FUNCTION_BLOCK goToRelPos (* Composite Function Block Type *)
  (* Standard: 61499-2 *)
  (* Version 1.0, 2019-05-27, Promok *)
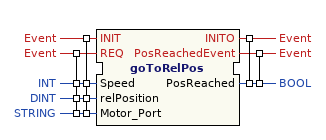
  EVENT_INPUT
    INIT WITH Speed, Motor_Port, relPosition; (* Initialization Request *)
    REQ WITH Speed, Motor_Port, relPosition; (* Normal Execution Request *)
  END_EVENT
  EVENT_OUTPUT
    INITO WITH PosReached; (* Initialization Confirm *)
    PosReachedEvent WITH PosReached;
  END_EVENT
  VAR_INPUT
    Speed : INT;
    relPosition : DINT;
    Motor_Port : STRING;
  END_VAR
  VAR_OUTPUT
    PosReached : BOOL;
  END_VAR
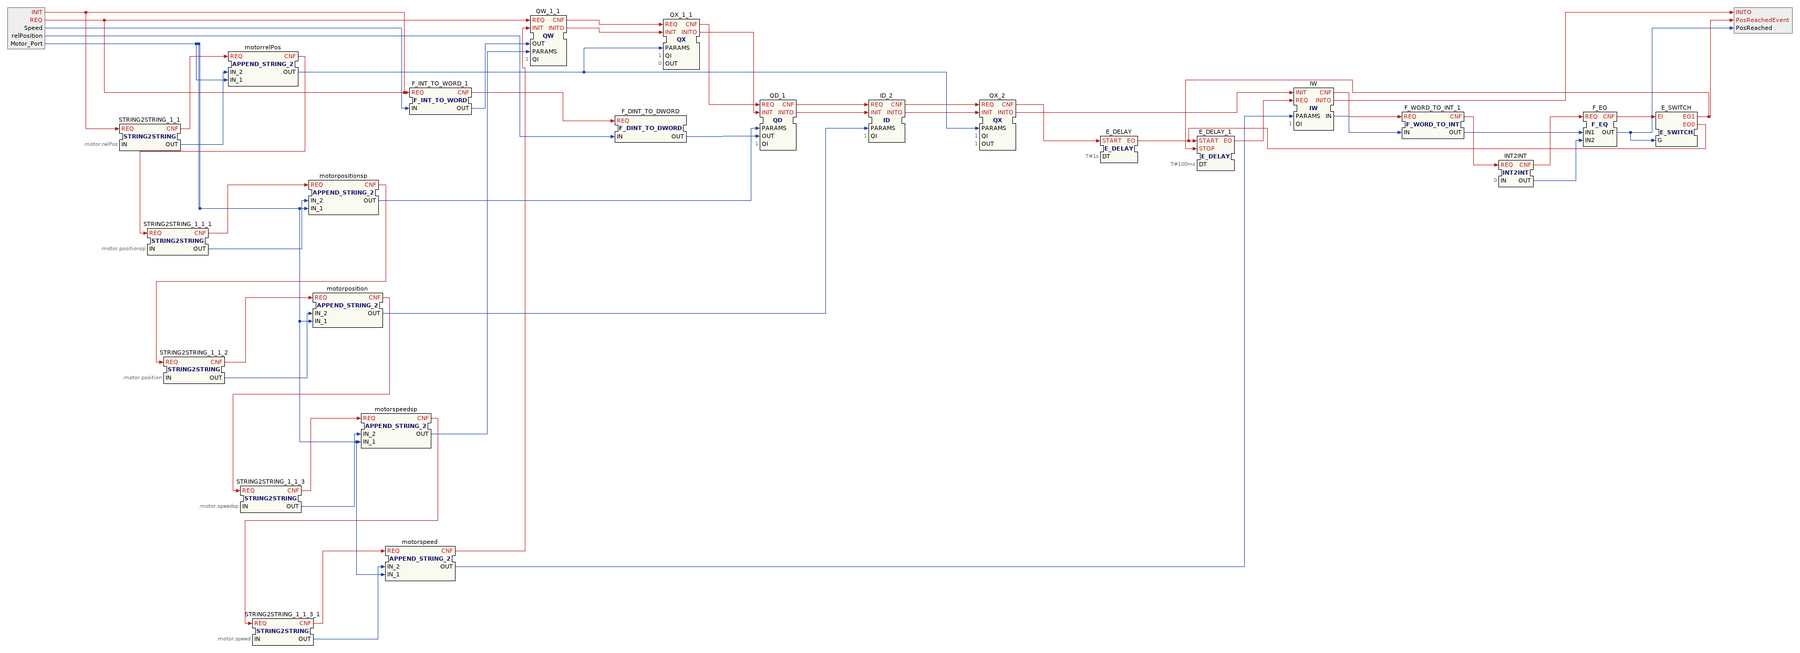
  FBS
    QX_1_1 : QX(QI := 1, OUT := 0);
    QW_1_1 : QW(QI := 1);
    QD_1 : QD(QI := 1);
    F_INT_TO_WORD_1 : F_INT_TO_WORD;
    ID_2 : ID(QI := 1);
    QX_2 : QX(QI := 1, OUT := 1);
    STRING2STRING_1_1 : STRING2STRING(IN := .motor.relPos);
    motorrelPos : APPEND_STRING_2;
    STRING2STRING_1_1_1 : STRING2STRING(IN := .motor.positionsp);
    motorpositionsp : APPEND_STRING_2;
    STRING2STRING_1_1_2 : STRING2STRING(IN := .motor.position);
    motorposition : APPEND_STRING_2;
    STRING2STRING_1_1_3 : STRING2STRING(IN := .motor.speedsp);
    motorspeedsp : APPEND_STRING_2;
    F_DINT_TO_DWORD : F_DINT_TO_DWORD;
    STRING2STRING_1_1_3_1 : STRING2STRING(IN := .motor.speed);
    motorspeed : APPEND_STRING_2;
    IW : IW(QI := 1);
    F_WORD_TO_INT_1 : F_WORD_TO_INT;
    E_DELAY : E_DELAY(DT := T#1s);
    F_EQ : F_EQ;
    INT2INT : INT2INT(IN := 0);
    E_SWITCH : E_SWITCH;
    E_DELAY_1 : E_DELAY(DT := T#100ms);
  END_FBS
  EVENT_CONNECTIONS
    QW_1_1.CNF TO QX_1_1.REQ;
    QW_1_1.INITO TO QX_1_1.INIT;
    QD_1.CNF TO ID_2.REQ;
    QX_1_1.CNF TO QD_1.REQ;
    QX_1_1.INITO TO QD_1.INIT;
    QD_1.INITO TO ID_2.INIT;
    STRING2STRING_1_1.CNF TO motorrelPos.REQ;
    STRING2STRING_1_1_1.CNF TO motorpositionsp.REQ;
    STRING2STRING_1_1_2.CNF TO motorposition.REQ;
    INIT TO STRING2STRING_1_1.REQ;
    motorrelPos.CNF TO STRING2STRING_1_1_1.REQ;
    motorpositionsp.CNF TO STRING2STRING_1_1_2.REQ;
    STRING2STRING_1_1_3.CNF TO motorspeedsp.REQ;
    motorposition.CNF TO STRING2STRING_1_1_3.REQ;
    REQ TO F_INT_TO_WORD_1.REQ;
    REQ TO QW_1_1.REQ;
    INIT TO F_INT_TO_WORD_1.REQ;
    F_INT_TO_WORD_1.CNF TO F_DINT_TO_DWORD.REQ;
    motorspeed.CNF TO QW_1_1.INIT;
    motorspeedsp.CNF TO STRING2STRING_1_1_3_1.REQ;
    STRING2STRING_1_1_3_1.CNF TO motorspeed.REQ;
    IW.CNF TO F_WORD_TO_INT_1.REQ;
    F_WORD_TO_INT_1.CNF TO INT2INT.REQ;
    INT2INT.CNF TO F_EQ.REQ;
    QX_2.CNF TO E_DELAY.START;
    ID_2.CNF TO QX_2.REQ;
    ID_2.INITO TO QX_2.INIT;
    IW.INITO TO INITO;
    QX_2.INITO TO IW.INIT;
    F_EQ.CNF TO E_SWITCH.EI;
    E_SWITCH.EO1 TO PosReachedEvent;
    E_DELAY.EO TO E_DELAY_1.START;
    E_DELAY_1.EO TO IW.REQ;
    E_SWITCH.EO1 TO E_DELAY_1.STOP;
    E_SWITCH.EO0 TO E_DELAY_1.START;
  END_CONNECTIONS
  DATA_CONNECTIONS
    F_INT_TO_WORD_1.OUT TO QW_1_1.OUT;
    STRING2STRING_1_1.OUT TO motorrelPos.IN_2;
    STRING2STRING_1_1_1.OUT TO motorpositionsp.IN_2;
    STRING2STRING_1_1_2.OUT TO motorposition.IN_2;
    Motor_Port TO motorrelPos.IN_1;
    Motor_Port TO motorpositionsp.IN_1;
    Motor_Port TO motorposition.IN_1;
    STRING2STRING_1_1_3.OUT TO motorspeedsp.IN_2;
    Motor_Port TO motorspeedsp.IN_1;
    motorspeedsp.OUT TO QW_1_1.PARAMS;
    motorrelPos.OUT TO QX_1_1.PARAMS;
    motorpositionsp.OUT TO QD_1.PARAMS;
    motorrelPos.OUT TO QX_2.PARAMS;
    motorposition.OUT TO ID_2.PARAMS;
    F_DINT_TO_DWORD.OUT TO QD_1.OUT;
    relPosition TO F_DINT_TO_DWORD.IN;
    Speed TO F_INT_TO_WORD_1.IN;
    STRING2STRING_1_1_3_1.OUT TO motorspeed.IN_2;
    Motor_Port TO motorspeed.IN_1;
    IW.IN TO F_WORD_TO_INT_1.IN;
    F_WORD_TO_INT_1.OUT TO F_EQ.IN1;
    motorspeed.OUT TO IW.PARAMS;
    INT2INT.OUT TO F_EQ.IN2;
    F_EQ.OUT TO PosReached;
    F_EQ.OUT TO E_SWITCH.G;
  END_CONNECTIONS
END_FUNCTION_BLOCK
